Fanuc TP program (LS listing): RET_HOME_STA60.LS

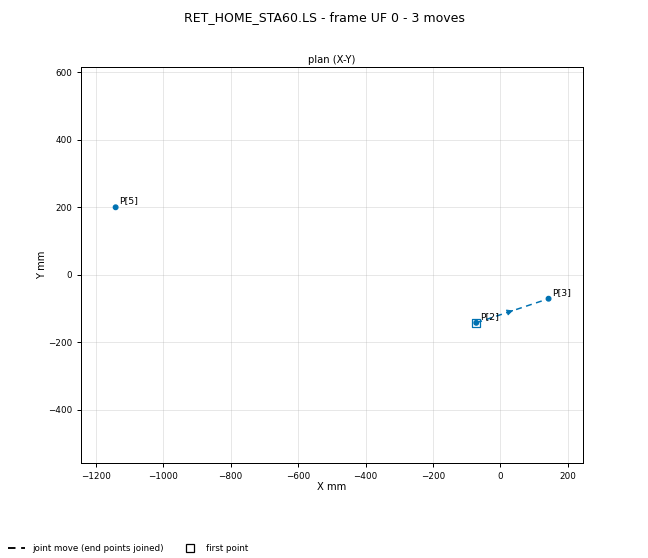
[picture p0: tool path of RET_HOME_STA60.LS in frame UF 0, 3 of 5 moves have a stored position in this frame; points joined in program order, loops and branches not executed]
/PROG  RET_HOME_STA60
/ATTR
OWNER		= SHIFT;
COMMENT		= "STA60 Return";
PROG_SIZE	= 1145;
CREATE		= DATE 18-11-04  TIME 07:33:20;
MODIFIED	= DATE 18-11-04  TIME 07:33:20;
FILE_NAME	= ARET_HOM;
VERSION		= 0;
LINE_COUNT	= 25;
MEMORY_SIZE	= 1417;
PROTECT		= READ_WRITE;
STORAGE		= SHADOW;
TCD:  STACK_SIZE	= 0,
      TASK_PRIORITY	= 50,
      TIME_SLICE	= 0,
      BUSY_LAMP_OFF	= 0,
      ABORT_REQUEST	= 0,
      PAUSE_REQUEST	= 0;
DEFAULT_GROUP	= 1,*,*,*,*;
CONTROL_CODE	= 00000000 00000000;
/APPL
  HANDLING : TRUE ;
/MN
   1:  !******************************** ;
   2:  !PATH: return home from ;
   3:  !        STA60 tool stands ;
   4:  !******************************** ;
   5:  !* ROBOT ID: IM01R02B02 ;
   6:  !*    F-196844 ;
   7:  !* Line: Line B02 ;
   8:  !******************************** ;
   9:   ;
  10:  UFRAME_NUM=0 ;
  11:  UTOOL_NUM=14 ;
  12:   ;
  13:  ENTER I-ZONE(2) ;
  14:  ENTER I-ZONE(1) ;
  15:   ;
  16:J P[1] 50% CNT100    ;
  17:J P[2] 50% CNT100    ;
  18:J P[3] 50% CNT100    ;
  19:J P[4] 50% CNT100    ;
  20:J P[5] 100% CNT100    ;
  21:   ;
  22:  EXIT I-ZONE(1) ;
  23:  EXIT I-ZONE(2) ;
  24:   ;
  25:  END ;
/POS
P[1]{
   GP1:
	UF : 0, UT : 14,
	J1=  -144.853 deg,	J2=   -28.708 deg,	J3=    82.000 deg,
	J4=     2.573 deg,	J5=   -83.800 deg,	J6=   -90.000 deg
};
P[2]{
   GP1:
	UF : 0, UT : 14,		CONFIG : 'N U B, 0, 0, 0',
	X =   -71.737  mm,	Y =  -142.116  mm,	Z =  2741.103  mm,
	W =   -91.792 deg,	P =     -.357 deg,	R =  -179.914 deg
};
P[3]{
   GP1:
	UF : 0, UT : 14,		CONFIG : 'N U B, 0, 0, 0',
	X =   142.665  mm,	Y =   -70.640  mm,	Z =  2741.103  mm,
	W =   -91.792 deg,	P =     -.357 deg,	R =   -89.472 deg
};
P[4]{
   GP1:
	UF : 0, UT : 14,
	J1=    95.076 deg,	J2=   -28.708 deg,	J3=    75.000 deg,
	J4=     2.573 deg,	J5=   -83.800 deg,	J6=   -90.000 deg
};
P[5]{
   GP1:
	UF : 0, UT : 14,		CONFIG : 'N U T, 0, 0, 0',
	X = -1140.855  mm,	Y =   200.393  mm,	Z =  2745.507  mm,
	W =   -98.230 deg,	P =    -1.434 deg,	R =    83.330 deg
};
/END
